Yaskawa INFORM job: TEST.JBI

/JOB
//NAME TEST
//INST
///ATTR SC,RW
///GROUP1 RB1
NOP
END
